INTERFACE I_CommonComponent EXTENDS I_ComponentBase

END_INTERFACE

(* stored: Version 1.1.0.1, ProductVersion 3.1.4024.12
   Itf I_CommonComponent: Id {5524175d-a60e-4641-b792-c92b917ff8cb} *)
